// Mitsubishi GX Works2 project: 0702   PLC: Q03UDV

// global labels: Global1
VAR_GLOBAL
  공급후진리드 AT X20 : BOOL;
  공급전진리드 AT X21 : BOOL;
  매거진센서 AT X22 : BOOL;
  고주파센서 AT X23 : BOOL;
  용량형센서 AT X24 : BOOL;
  근접포토센서 AT X25 : BOOL;
  그리퍼온리드 AT X27 : BOOL;
  그리퍼오프리드 AT X28 : BOOL;
  물품도착포토 AT X29 : BOOL;
  TG1 AT X2A : BOOL;
  TG2 AT X2B : BOOL;
  TG3 AT X2C : BOOL;
  PB4 AT X2D : BOOL;
  PB5 AT X2E : BOOL;
  창고1 AT X30 : BOOL;
  창고2 AT X31 : BOOL;
  창고3 AT X32 : BOOL;
  창고4 AT X33 : BOOL;
  창고5 AT X34 : BOOL;
  창고6 AT X35 : BOOL;
  창고7 AT X36 : BOOL;
  창고8 AT X37 : BOOL;
  창고9 AT X38 : BOOL;
  도어센서 AT X39 : BOOL;
  압력센서 AT X3A : BOOL;
  공급전솔 AT Y40 : BOOL;
  공급후솔 AT Y41 : BOOL;
  그리퍼온솔 AT Y42 : BOOL;
  그리퍼오프솔 AT Y43 : BOOL;
  경광녹색 AT Y44 : BOOL;
  경광황색 AT Y45 : BOOL;
  경광적색 AT Y46 : BOOL;
  부저 AT Y47 : BOOL;
  컨베이어 AT Y48 : BOOL;
  램프1 AT Y4A : BOOL;
  램프2 AT Y4B : BOOL;
  램프3 AT Y4C : BOOL;
  램프5 AT Y4D : BOOL;
  램프4 AT Y4E : BOOL;
  R그립온명령 AT X1000 : BOOL;
  R그립오프명령 AT X1001 : BOOL;
  R_PLC시작 AT X1002 : BOOL;
  R_판별리셋 AT X1003 : BOOL;
  R재공급 AT X1004 : BOOL;
  R그립온센서 AT Y1000 : BOOL;
  R그립오프센서 AT Y1001 : BOOL;
  R물품없음 AT Y1002 : BOOL;
  R_금속 AT Y1003 : BOOL;
  R_검비금속 AT Y1004 : BOOL;
  R_흰비금속 AT Y1005 : BOOL;
  R물품도착 AT Y1006 : BOOL;
  R컨베이어 AT Y1007 : BOOL;
  R_재시작 AT Y1008 : BOOL;
  R_interrupt AT Y1009 : BOOL;
  R창고1 AT Y100A : BOOL;
  R창고2 AT Y100B : BOOL;
  R창고3 AT Y100C : BOOL;
  R창고4 AT Y100D : BOOL;
  R창고5 AT Y100E : BOOL;
  R창고6 AT Y100F : BOOL;
  R창고7 AT Y1010 : BOOL;
  R창고8 AT Y1011 : BOOL;
  R창고9 AT Y1012 : BOOL;
  R창고A AT Y1013 : BOOL;
END_VAR

PROGRAM MAIN
VAR
  T_매거진없음 : TIMER;
  공작물공급 : BOOL;
  작동중 : BOOL;
  비화 : BOOL;
  비금 : BOOL;
  금속 : BOOL;
  T_컨베이어 : TIMER;
  종료 : BOOL;
  컨정지 : BOOL;
  용량형탐지 : BOOL;
  고주파탐지 : BOOL;
  근접포토탐지 : BOOL;
  T도착지연 : TIMER;
  plc공정종료 : BOOL;
END_VAR
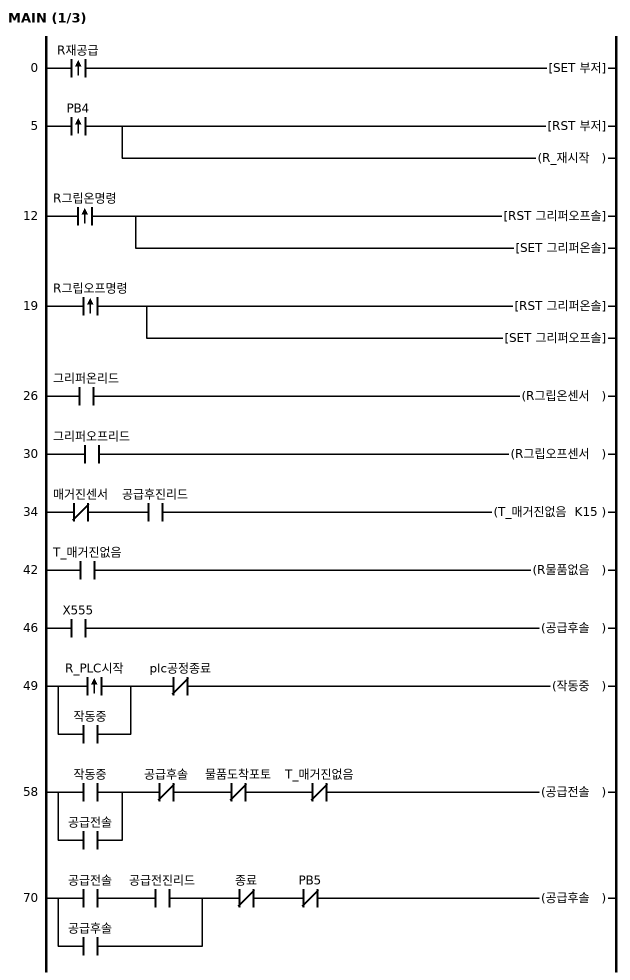
0     LDP     R재공급
      SET     부저
5     LDP     PB4
      RST     부저
      OUT     R_재시작
12    LDP     R그립온명령
      RST     그리퍼오프솔
      SET     그리퍼온솔
19    LDP     R그립오프명령
      RST     그리퍼온솔
      SET     그리퍼오프솔
26    LD      그리퍼온리드
      OUT     R그립온센서
30    LD      그리퍼오프리드
      OUT     R그립오프센서
34    LDI     매거진센서
      AND     공급후진리드
      OUT     T_매거진없음 K15
42    LD      T_매거진없음
      OUT     R물품없음
46    LD      X555
      OUT     공급후솔
49    LDP     R_PLC시작
      OR      작동중
      ANI     plc공정종료
      OUT     작동중
58    LD      작동중
      OR      공급전솔
      ANI     공급후솔
      ANI     물품도착포토
      ANI     T_매거진없음
      OUT     공급전솔
70    LD      공급전솔
      AND     공급전진리드
      OR      공급후솔
      ANI     종료
      ANI     PB5
      OUT     공급후솔
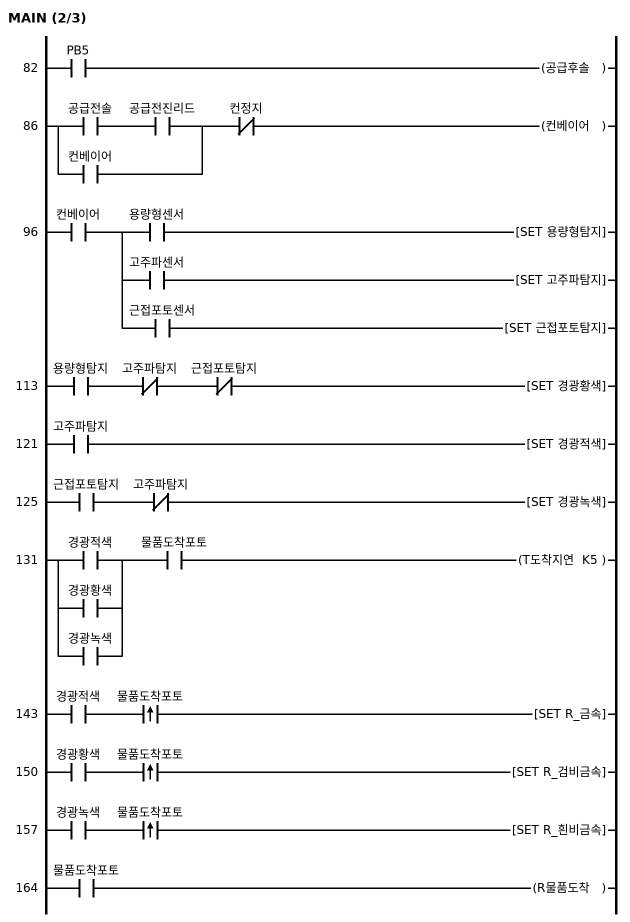
82    LD      PB5
      OUT     공급후솔
86    LD      공급전솔
      AND     공급전진리드
      OR      컨베이어
      ANI     컨정지
      OUT     컨베이어
96    LD      컨베이어
      MPS
      AND     용량형센서
      SET     용량형탐지
      MRD
      AND     고주파센서
      SET     고주파탐지
      MPP
      AND     근접포토센서
      SET     근접포토탐지
113   LD      용량형탐지
      ANI     고주파탐지
      ANI     근접포토탐지
      SET     경광황색
121   LD      고주파탐지
      SET     경광적색
125   LD      근접포토탐지
      ANI     고주파탐지
      SET     경광녹색
131   LD      경광적색
      OR      경광황색
      OR      경광녹색
      AND     물품도착포토
      OUT     T도착지연 K5
143   LD      경광적색
      ANDP    물품도착포토
      SET     R_금속
150   LD      경광황색
      ANDP    물품도착포토
      SET     R_검비금속
157   LD      경광녹색
      ANDP    물품도착포토
      SET     R_흰비금속
164   LD      물품도착포토
      OUT     R물품도착
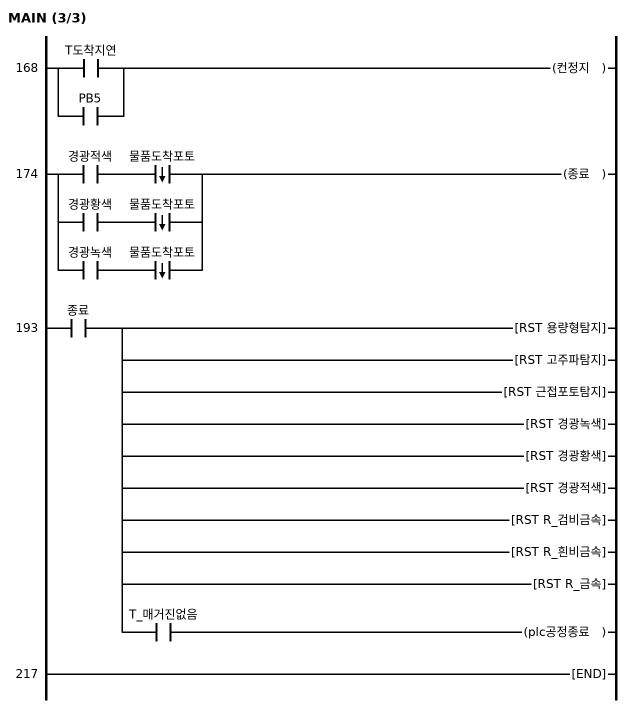
168   LD      T도착지연
      OR      PB5
      OUT     컨정지
174   LD      경광적색
      ANDF    물품도착포토
      LD      경광황색
      ANDF    물품도착포토
      ORB
      LD      경광녹색
      ANDF    물품도착포토
      ORB
      OUT     종료
193   LD      종료
      RST     용량형탐지
      RST     고주파탐지
      RST     근접포토탐지
      RST     경광녹색
      RST     경광황색
      RST     경광적색
      RST     R_검비금속
      RST     R_흰비금속
      RST     R_금속
      AND     T_매거진없음
      OUT     plc공정종료
217   END
END_PROGRAM
